{attribute 'qualified_only'}
{attribute 'strict'}
TYPE E_MbWordOrder :
(
	Inherit := 0,
	ABCD,
	CDAB,
	BADC,
	DCBA
);
END_TYPE

(* stored: Version 1.1.0.1
   DUT E_MbWordOrder: Id {dcaec71b-99c9-41be-ad1c-8f81d086eb70} *)
